// LS Electric XG5000 project: 물품보관함_최최종
// PLC LSPLC

PROGRAM NewProgram (task: 스캔 프로그램)

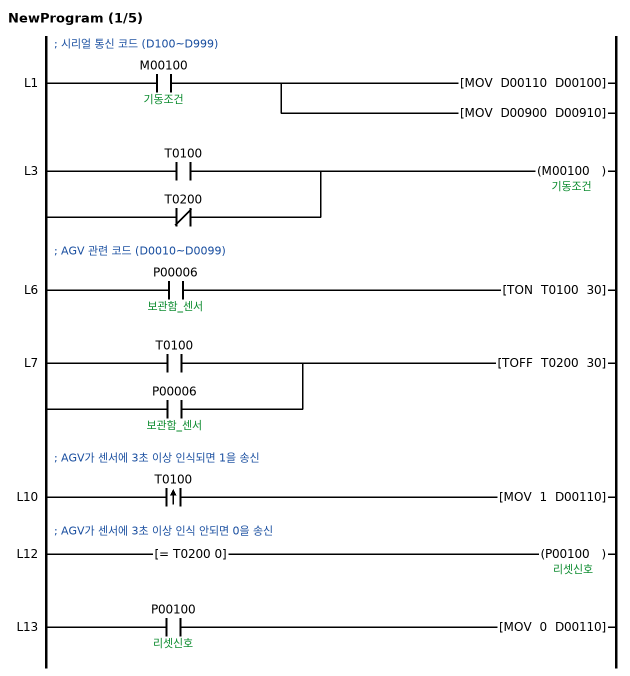
// 시리얼 통신 코드 (D100~D999)
; L1
LOAD      M00100	// 기동조건
MOV       D00110 D00100
MOV       D00900 D00910
; L3
LOAD      T0100
OR NOT    T0200
OUT       M00100	// 기동조건
// AGV 관련 코드 (D0010~D0099)
; L6
LOAD      P00006	// 보관함_센서
TON       T0100 30
; L7
LOAD      T0100
OR        P00006	// 보관함_센서
TOFF      T0200 30
// AGV가 센서에 3초 이상 인식되면 1을 송신
; L10
LOADP     T0100
MOV       1 D00110
// AGV가 센서에 3초 이상 인식 안되면 0을 송신
; L12
LOAD=     T0200 0
OUT       P00100	// 리셋신호
; L13
LOAD      P00100	// 리셋신호
MOV       0 D00110

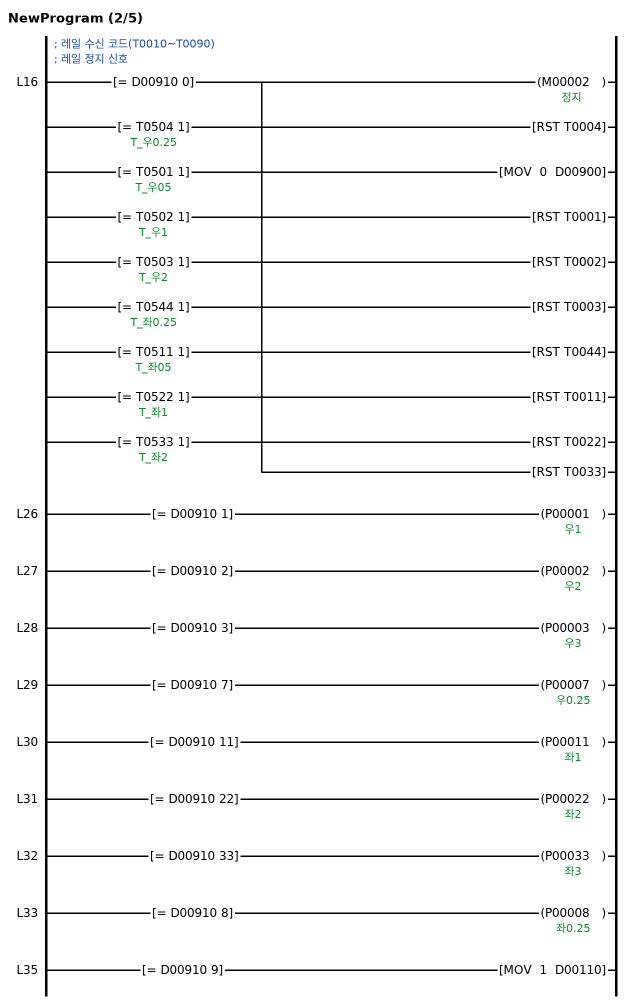
// 레일 수신 코드(T0010~T0090)
// 레일 정지 신호
; L16
LOAD=     D00910 0
OR=       T0504 1	// T_우0.25
OR=       T0501 1	// T_우05
OR=       T0502 1	// T_우1
OR=       T0503 1	// T_우2
OR=       T0544 1	// T_좌0.25
OR=       T0511 1	// T_좌05
OR=       T0522 1	// T_좌1
OR=       T0533 1	// T_좌2
OUT       M00002	// 정지
RST       T0004
MOV       0 D00900
RST       T0001
RST       T0002
RST       T0003
RST       T0044
RST       T0011
RST       T0022
RST       T0033
; L26
LOAD=     D00910 1
OUT       P00001	// 우1
; L27
LOAD=     D00910 2
OUT       P00002	// 우2
; L28
LOAD=     D00910 3
OUT       P00003	// 우3
; L29
LOAD=     D00910 7
OUT       P00007	// 우0.25
; L30
LOAD=     D00910 11
OUT       P00011	// 좌1
; L31
LOAD=     D00910 22
OUT       P00022	// 좌2
; L32
LOAD=     D00910 33
OUT       P00033	// 좌3
; L33
LOAD=     D00910 8
OUT       P00008	// 좌0.25
; L35
LOAD=     D00910 9
MOV       1 D00110

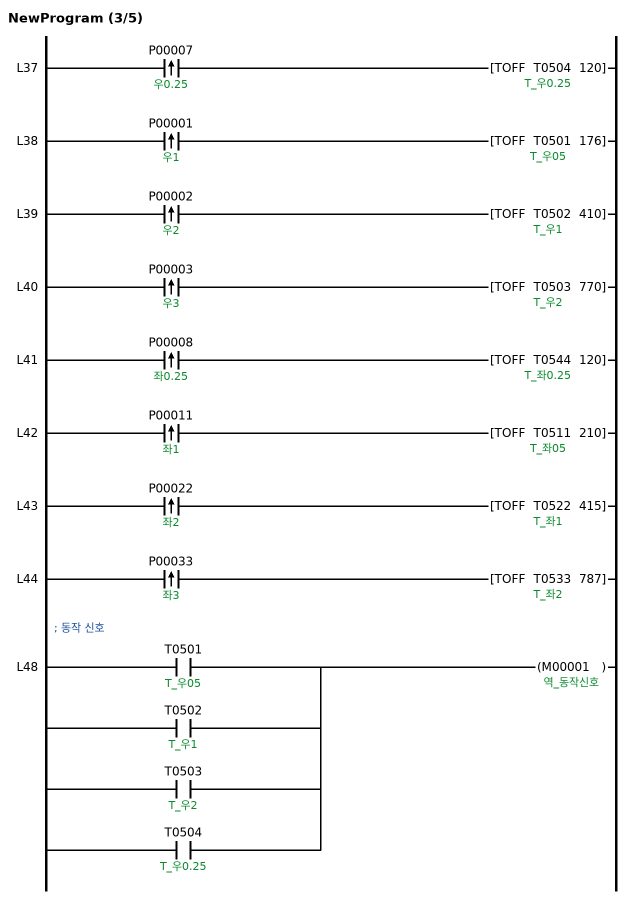
; L37
LOADP     P00007	// 우0.25
TOFF      T0504 120	// T_우0.25
; L38
LOADP     P00001	// 우1
TOFF      T0501 176	// T_우05
; L39
LOADP     P00002	// 우2
TOFF      T0502 410	// T_우1
; L40
LOADP     P00003	// 우3
TOFF      T0503 770	// T_우2
; L41
LOADP     P00008	// 좌0.25
TOFF      T0544 120	// T_좌0.25
; L42
LOADP     P00011	// 좌1
TOFF      T0511 210	// T_좌05
; L43
LOADP     P00022	// 좌2
TOFF      T0522 415	// T_좌1
; L44
LOADP     P00033	// 좌3
TOFF      T0533 787	// T_좌2
// 동작 신호
; L48
LOAD      T0501	// T_우05
OR        T0502	// T_우1
OR        T0503	// T_우2
OR        T0504	// T_우0.25
OUT       M00001	// 역_동작신호

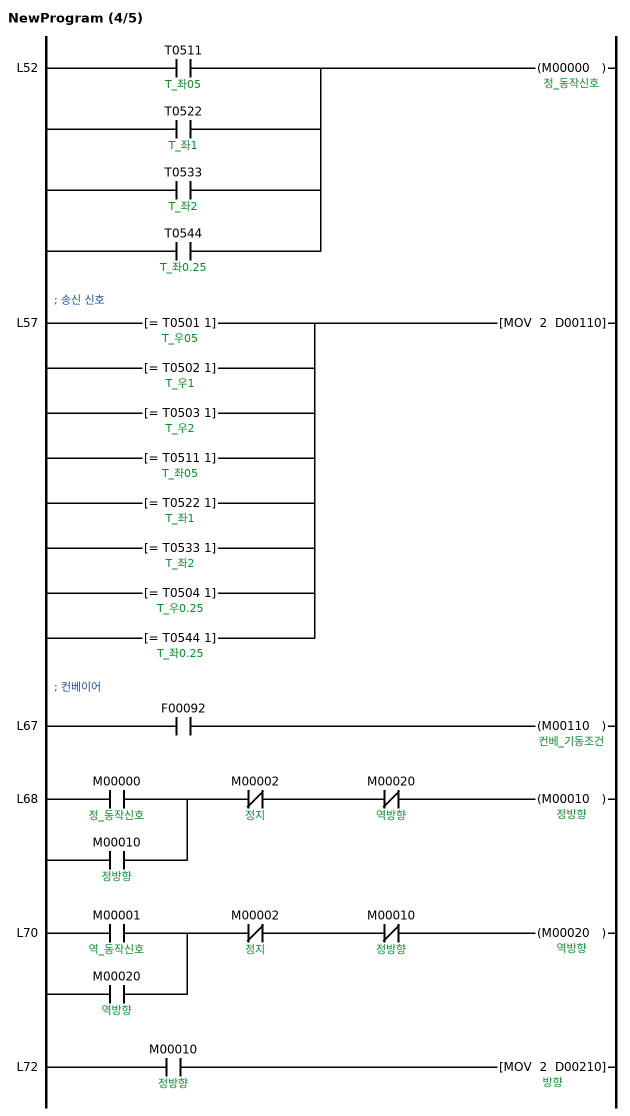
; L52
LOAD      T0511	// T_좌05
OR        T0522	// T_좌1
OR        T0533	// T_좌2
OR        T0544	// T_좌0.25
OUT       M00000	// 정_동작신호
// 송신 신호
; L57
LOAD=     T0501 1	// T_우05
OR=       T0502 1	// T_우1
OR=       T0503 1	// T_우2
OR=       T0511 1	// T_좌05
OR=       T0522 1	// T_좌1
OR=       T0533 1	// T_좌2
OR=       T0504 1	// T_우0.25
OR=       T0544 1	// T_좌0.25
MOV       2 D00110
// 컨베이어
; L67
LOAD      F00092
OUT       M00110	// 컨베_기동조건
; L68
LOAD      M00000	// 정_동작신호
OR        M00010	// 정방향
AND NOT   M00002	// 정지
AND NOT   M00020	// 역방향
OUT       M00010	// 정방향
; L70
LOAD      M00001	// 역_동작신호
OR        M00020	// 역방향
AND NOT   M00002	// 정지
AND NOT   M00010	// 정방향
OUT       M00020	// 역방향
; L72
LOAD      M00010	// 정방향
MOV       2 D00210	// 방향

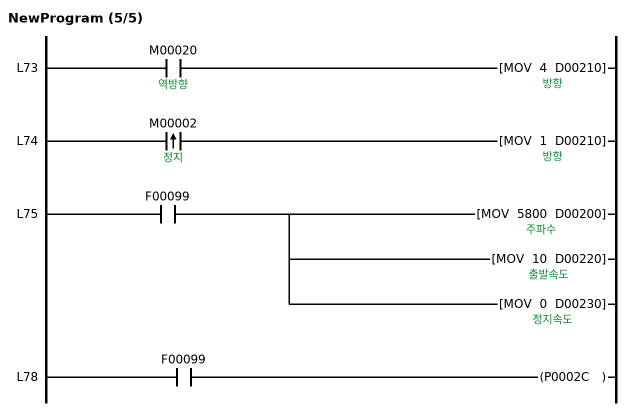
; L73
LOAD      M00020	// 역방향
MOV       4 D00210	// 방향
; L74
LOADP     M00002	// 정지
MOV       1 D00210	// 방향
; L75
LOAD      F00099
MOV       5800 D00200	// 주파수
MOV       10 D00220	// 출발속도
MOV       0 D00230	// 정지속도
; L78
LOAD      F00099
OUT       P0002C

VARIABLES AND COMMENTS (devices not used above)
P00004	BIT	AGV_센서
P00020	BIT	대기신호